Xinje XDPPro project, PLC1: XDH-60T4 (software 3.7.4b 2021-06-17)

PROGRAM Ladder

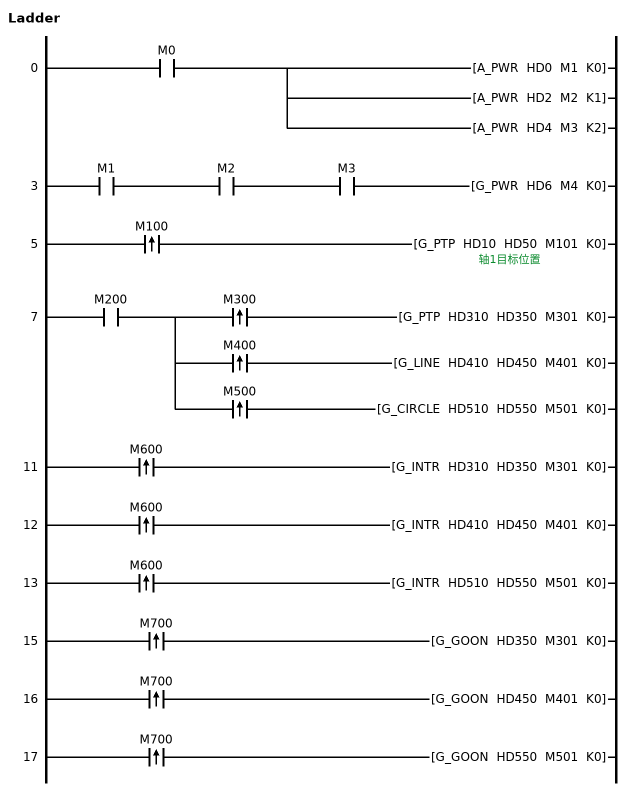
LD     M0
A_PWR  HD0 M1 K0
A_PWR  HD2 M2 K1
A_PWR  HD4 M3 K2
LD     M1
AND    M2
AND    M3
G_PWR  HD6 M4 K0
LDP    M100
G_PTP  HD10 HD50 M101 K0	; 轴1目标位置
LD     M200
MPS
ANDP   M300
G_PTP  HD310 HD350 M301 K0
MRD
ANDP   M400
G_LINE HD410 HD450 M401 K0
MPP
ANDP   M500
G_CIRCLE HD510 HD550 M501 K0
LDP    M600
G_INTR HD310 HD350 M301 K0
LDP    M600
G_INTR HD410 HD450 M401 K0
LDP    M600
G_INTR HD510 HD550 M501 K0
LDP    M700
G_GOON HD350 M301 K0
LDP    M700
G_GOON HD450 M401 K0
LDP    M700
G_GOON HD550 M501 K0

COMMENTS (devices not used above)
D20444	轴3当前位置
D20244	轴2当前位置
HD100	轴0目标绝对位置
HD200	轴1目标绝对位置
D20044	轴1当前位置
HD14	轴2目标位置
HD18	轴3目标位置

C FUNCTION BLOCK func1.fcb
/*************************************************************************
   FunctionBlockName:  FUNC1
   Version:            1.0.0
   Author:             
   UpdateTime:         2021-08-21 17:10:53
   Comment:            
			
**************************************************************************/
void FUNC1( WORD W , BIT B )
{
#define SysRegAddr_HD_D_HM_M
#define DFHD *(FP64*)&HD

HD[100] = 6;            //数据行数
HD[101] = 0;            //0：继续插入 1：重新装载

HD[110] = 1;            //行号1
HD[112] = 1;            //类型：line
HD[113] = 0;            //参数
DFHD[116] = 100000;     //目标X
DFHD[120] = 100000;     //目标Y
DFHD[124] = 0;          //目标Z
DFHD[164] = 20000;      //目标速度

HD[170] = 2;            //行号2
HD[172] = 0;            //类型：PTP
HD[173] = 0;            //参数
DFHD[176] = 200000;     //目标X
DFHD[180] = 150000;     //目标Y
DFHD[184] = 0;          //目标Z
DFHD[224] = 20000;      //目标速度

HD[230] = 3;            //行号3
HD[232] = 0;            //类型
HD[233] = 0;            //参数
DFHD[236] = 100000;     //目标X
DFHD[240] = 400000;     //目标Y
DFHD[244] = 0;          //目标Z
DFHD[284] = 20000;      //目标速度

HD[290] = 4;            //行号4
HD[292] = 1;            //类型：line
HD[293] = 0;            //参数
DFHD[296] = 0;          //目标X
DFHD[300] = 0;          //目标Y
DFHD[304] = 0;          //目标Z
DFHD[344] = 20000;      //目标速度


HD[350] = 5;            //行号5
HD[352] = 2;            //类型：circle
HD[353] = 0;            //参数
DFHD[356] = 30000;      //目标X
DFHD[360] = 100000;          //目标Y
DFHD[364] = 0;          //目标Z
DFHD[380] = 50000;      //辅助X
DFHD[384] = 25000;      //辅助Y
DFHD[388] = 0;          //辅助Z
DFHD[404] = 20000;      //目标速度

/*
HD[350] = 5;            //行号5
HD[352] = 200;          //类型
HD[353] = 0;            //参数
*/

HD[410] = 6;            //行号6
HD[412] = 200;          //类型
HD[413] = 0;            //参数
}